TYPE T_Ctrl_SIf_ICL :
STRUCT
	///configuration
	Cfg: T_Ctrl_SIf_ICL_Cfg;
	///parameter
	Par: T_Ctrl_SIf_ICL_Par;
	///current values
	Cur: T_Ctrl_SIf_ICL_Cur;
	///io input
	In: T_Ctrl_SIf_ICL_In;
END_STRUCT
END_TYPE

(* stored: Version 1.1.0.1, ProductVersion 3.1.0.19
   DUT T_Ctrl_SIf_ICL: Id {9967b90c-d64b-496b-b364-92b073b4403a} *)
